(*
SPDX-FileCopyrightText: Â© 2026 Oleksandr Tiutyk <trofimich@gmail.com>
SPDX-License-Identifier: MIT
License: https://opensource.org/license/mit
*)

(*!
<summary>Configuration and control contract for an analog output component.</summary>
<description>
Extends IReadOnlyAnalogOutput with hardware IO binding methods and value mutator.
</description>
*)

INTERFACE IAnalogOutput EXTENDS IReadOnlyAnalogOutput

(*!
<summary>Binds component to a 16-bit signed integer output process image variable '%Q*'.</summary>
<param name="rawVariable">Reference to physical INT output variable.</param>
*)
METHOD BindToInt16IO
VAR_INPUT
	rawVariable : REFERENCE TO INT;
END_VAR
END_METHOD

(*!
<summary>Binds component to a 32-bit signed integer output process image variable '%Q*'.</summary>
<param name="rawVariable">Reference to physical DINT output variable.</param>
*)
METHOD BindToInt32IO
VAR_INPUT
	rawVariable : REFERENCE TO DINT;
END_VAR
END_METHOD

(*!
<summary>Binds component to a 32-bit float output process image variable '%Q*'.</summary>
<param name="rawVariable">Reference to physical REAL output variable.</param>
*)
METHOD BindToReal32IO
VAR_INPUT
	rawVariable : REFERENCE TO REAL;
END_VAR
END_METHOD

(*!
<summary>Gets or sets engineering unit value to output.</summary>
*)
{attribute 'monitoring' := 'call'}
PROPERTY Value : LREAL
GET
END_GET
SET
END_SET
END_PROPERTY

END_INTERFACE

(* stored: Version 1.1.0.1
   Itf IAnalogOutput: Id {9faf0717-a113-4ecb-80ad-8a4483a7a4ab}
   Method BindToInt16IO: Id {cfafbf5a-28a4-42b6-b6c8-02961a053799}
   Method BindToInt32IO: Id {7e02e96a-73e2-4dec-9e13-577ec603a62d}
   Method BindToReal32IO: Id {a4b5116f-4ebc-475d-b011-1b4cb4eacbde}
   Property Value: Id {3698dd6a-f924-4203-b3de-f32a2da4dc57}
   Get Get: Id {7d8b7e41-98a0-4948-a914-df63ea484367}
   Set Set: Id {7c70f7ee-324f-475c-803e-937de0b7d0e0} *)
